RoboDK station: AROB_AS3_A1_Vorlage.rdk

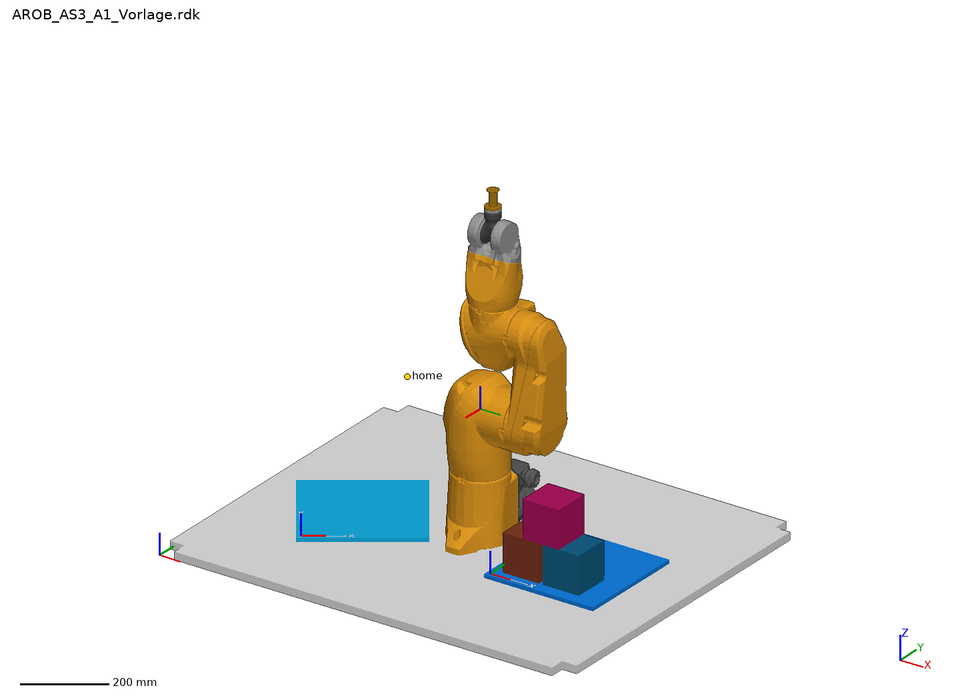
[picture v0: the station drawn from its stored meshes, robots at their saved joint values, targets as dots, program paths as lines]
Station AROB_AS3_A1 (saved by RoboDK 5.6.9). Poses are relative to the parent item; angles as X-Y-Z fixed-axis rotations.
  - frame world at (0, 0, 0) mm
    - frame Staubli TX2-40 Base at (560, 460, 340) mm, rotated rx 0 ry 0 rz -90 deg
      - robot Staubli TX2-40: 6 axes, payload 1.7 kg, reach 515 mm, repeatability 0.02 mm, weight 29 kg
          modified DH rows (alpha deg, a mm, theta deg, d mm): 0, 0, 0, 320; -90, 0, -90, 35; 0, 225, -90, 0; -90, 0, 0, 225; 90, 0, 0, 0; -90, 0, 180, 65
          base shift (0, 0, -320) mm
          joint limits [-180, -125, -138, -270, -120, -270] to [180, 125, 138, 270, 133.5, 270]; home [0, 0, 90, 0, 0, 0]; saved at [0, 0, 0, 0, 0, 0]
        - tool needle, TCP at (0, 0, 65) mm, size 40 x 40 x 65 mm, geometry from needle.iges
        - tool gripper, TCP at (0, 0, 45) mm, size 39.7 x 39.8 x 45 mm
    - object workspace_plate at (0, 0, 0) mm, size 1120 x 920 x 31 mm, geometry from workspace_plate.iges
    - target home (Cartesian target) at (595, 125, 565) mm, rotated rx 0 ry 90 rz -90 deg; joints [0, 0, 90, 0, 0, 0] of Staubli TX2-40
  - frame PickFrame at (240.25, 211.56, 31) mm, rotated rx 0 ry 0 rz 35.13 deg
  - frame PlaceFrame at (700, 300, 30) mm
    - object plate at (0, 0, 0) mm, size 300 x 300 x 11 mm, geometry from plate.iges
    - object cube3 at (180, 70, 50) mm, size 100 x 100 x 100 mm, geometry from cube.iges
    - object cube1 at (70, 70, 50) mm, size 100 x 100 x 100 mm, geometry from cube.iges
    - object cube2 at (125, 70, 150) mm, size 100 x 100 x 100 mm, geometry from cube.iges
  - Python program ProgPickPlace (listed below)
  - Python program ProgReset (listed below)

--- Python program ProgPickPlace ---
# Type help("robodk.robolink") or help("robodk.robomath") for more information
# Press F5 to run the script
# Documentation: https://robodk.com/doc/en/RoboDK-API.html
# Reference:     https://robodk.com/doc/en/PythonAPI/robodk.html
# Note: It is not required to keep a copy of this file, your Python script is saved with your RDK project

# You can also use the new version of the API:
import robodk.robolink as rl    # RoboDK API
import robodk.robomath as rm    # Robot toolbox
import math

RDK = rl.Robolink()

robot = RDK.Item("Staubli TX2-40")

world = RDK.Item("world")
pick_frame = RDK.Item("PickFrame")
place_frame = RDK.Item("PlaceFrame")
home = RDK.Item("home")

tool_gripper = RDK.Item("gripper")

#cubes =[RDK.Item("cube1"), RDK.Item("cube2"), RDK.Item("cube3")]
#cubes.sort(key=lambda x: x.Pose()[2,3], reverse=True)

robot.setSpeed(50, 50, 150, 150)

pick_list = [[ 70,70, 50,0,0,0], [180,70, 50,0,0,0], [125,70,150,0,0,0]]
pick_list.sort(key=lambda x: x[2], reverse=True)
place_list = pick_list

# go home, robot
for i in range(0,3):
    cube_pick_above = rm.Staubli_2_Pose(pick_list[i]) * rm.transl(0,0,120) * rm.rotx(math.radians(180))
    cube_pick_hit   = rm.Staubli_2_Pose(pick_list[i]) * rm.transl(0,0,48) * rm.rotx(math.radians(180))
    cube_pick_top   = rm.Staubli_2_Pose(pick_list[i]) * rm.transl(0,0,120)

    cube_place_above = rm.Staubli_2_Pose(pick_list[(len(place_list) - 1) - i]) * rm.transl(0,0,120) * rm.rotx(math.radians(180))
    cube_place_hit   = rm.Staubli_2_Pose(pick_list[(len(place_list) - 1) - i]) * rm.transl(0,0,48) * rm.rotx(math.radians(180))
    cube_place_top   = rm.Staubli_2_Pose(pick_list[(len(place_list) - 1) - i]) * rm.transl(0,0,120)


    robot.setFrame(pick_frame)
    robot.MoveJ(cube_pick_above) # move over block
    robot.MoveL(cube_pick_hit) # plung into block
    robot.MoveL(cube_pick_hit * rm.transl(0,0,2)) # realism
    tool_gripper.AttachClosest()
    robot.MoveL(cube_pick_above) # move back up

    robot.setPoseFrame(world)
    robot.MoveJ(home) # go home

    robot.setPoseFrame(place_frame)
    robot.MoveJ(cube_place_above) # move over block
    robot.MoveL(cube_place_hit) # plung into block
    robot.MoveL(cube_place_hit * rm.transl(0,0,2)) # realism
    tool_gripper.DetachAll(parent=place_frame)
    robot.MoveL(cube_place_above) # move back up

    robot.setPoseFrame(world)
    robot.MoveJ(home) # go home

--- Python program ProgReset ---
# Type help("robodk.robolink") or help("robodk.robomath") for more information
# Press F5 to run the script
# Documentation: https://robodk.com/doc/en/RoboDK-API.html
# Reference:     https://robodk.com/doc/en/PythonAPI/robodk.html
# Note: It is not required to keep a copy of this file, your Python script is saved with your RDK project

# You can also use the new version of the API:
import robodk.robomath as rm
import robodk.robolink as rl

RDK = rl.Robolink()

robot = RDK.Item("Staubli TX2-40")
world = RDK.Item("world")
pick_frame = RDK.Item("PickFrame")
place_frame = RDK.Item("PlaceFrame")
home = RDK.Item("home")
tool_gripper = RDK.Item("gripper")

# go home, robot
robot.setPoseFrame(world)
robot.MoveJ(home)
tool_gripper.DetachAll()

cubes =[RDK.Item("cube1"), RDK.Item("cube2"), RDK.Item("cube3")]

cubes[0].setParent(pick_frame)
cubes[0].setPose(rm.Staubli_2_Pose([ 70,70, 50,0,0,0]))
cubes[1].setParent(pick_frame)
cubes[1].setPose(rm.Staubli_2_Pose([180,70, 50,0,0,0]))
cubes[2].setParent(pick_frame)
cubes[2].setPose(rm.Staubli_2_Pose([125,70,150,0,0,0]))
